LIN {X 0,Y 179.464,Z 996.724,A -85,B 0,C 180,E1 20811.906,E2 20811.906} C_VEL
LIN {X 0,Y 188.427,Z 983.505,A -85,B 0,C 180,E1 20823.22,E2 20823.22} C_VEL
LIN {X 0,Y 202.809,Z 964.358,A -85,B 0,C 180,E1 20832.94,E2 20832.94} C_VEL
LIN {X 0,Y 221.661,Z 939.292,A -85,B 0,C 180,E1 20840.906,E2 20840.906} C_VEL
LIN {X 0,Y 224.713,Z 937.25,A -85,B 0,C 180,E1 20842.19,E2 20842.19} C_VEL
LIN {X 0,Y 206.607,Z 940.656,A -85,B 0,C 180,E1 20849.15,E2 20849.15} C_VEL
LIN {X 0,Y 193.54,Z 940.036,A -85,B 0,C 180,E1 20856.986,E2 20856.986} C_VEL
LIN {X 0,Y 184.714,Z 935.319,A -85,B 0,C 180,E1 20865.776,E2 20865.776} C_VEL
LIN {X 0,Y 180.026,Z 924.585,A -85,B 0,C 180,E1 20876.395,E2 20876.395} C_VEL
LIN {X 0,Y 191.865,Z 914.932,A -85,B 0,C 180,E1 20893.704,E2 20893.704} C_VEL
LIN {X 0,Y 212.483,Z 904.44,A -85,B 0,C 180,E1 20904.008,E2 20904.008} C_VEL
LIN {X 0,Y 233.891,Z 893.022,A -85,B 0,C 180,E1 20910.12,E2 20910.12} C_VEL
LIN {X 0,Y 248.033,Z 884.252,A -85,B 0,C 180,E1 20912.881,E2 20912.881} C_VEL
LIN {X 0,Y 238.457,Z 902.02,A -85,B 0,C 180,E1 20915.584,E2 20915.584} C_VEL
LIN {X 0,Y 228.286,Z 914.831,A -85,B 0,C 180,E1 20917.177,E2 20917.177} C_VEL
LIN {X 0,Y 217.808,Z 926.758,A -85,B 0,C 180,E1 20919.046,E2 20919.046} C_VEL
LIN {X 0,Y 200.214,Z 949.54,A -85,B 0,C 180,E1 20926.435,E2 20926.435} C_VEL
LIN {X 0,Y 185.842,Z 966.385,A -85,B 0,C 180,E1 20935.229,E2 20935.229} C_VEL
LIN {X 0,Y 174.431,Z 979.636,A -85,B 0,C 180,E1 20947.008,E2 20947.008} C_VEL
LIN {X 0,Y 169.075,Z 986.655,A -85,B 0,C 180,E1 20959.683,E2 20959.683} C_VEL
LIN {X 0,Y 168.279,Z 988.372,A -85,B 0,C 180,E1 20970.001,E2 20970.001} C_VEL
LIN {X 0,Y 169.698,Z 985.642,A -85,B 0,C 180,E1 20982.889,E2 20982.889} C_VEL
LIN {X 0,Y 176.265,Z 977.344,A -85,B 0,C 180,E1 20995.436,E2 20995.436} C_VEL
LIN {X 0,Y 188.345,Z 963.517,A -85,B 0,C 180,E1 21006.483,E2 21006.483} C_VEL
LIN {X 0,Y 204.243,Z 944.465,A -85,B 0,C 180,E1 21015.398,E2 21015.398} C_VEL
LIN {X 0,Y 221.705,Z 921.014,A -85,B 0,C 180,E1 21022.202,E2 21022.202} C_VEL
LIN {X 0,Y 239.619,Z 892.347,A -85,B 0,C 180,E1 21027.459,E2 21027.459} C_VEL
LIN {X 0,Y 247.476,Z 877.194,A -85,B 0,C 180,E1 21029.455,E2 21029.455} C_VEL
LIN {X 0,Y 247.461,Z 861.301,A -85,B 0,C 180,E1 21034.633,E2 21034.633} C_VEL
LIN {X 0,Y 245.563,Z 845.485,A -85,B 0,C 180,E1 21041.277,E2 21041.277} C_VEL
LIN {X 0,Y 243.44,Z 835.366,A -85,B 0,C 180,E1 21047.419,E2 21047.419} C_VEL
LIN {X 0,Y 242.204,Z 826.553,A -85,B 0,C 180,E1 21056.408,E2 21056.408} C_VEL
LIN {X 0,Y 242.269,Z 825.858,A -85,B 0,C 180,E1 21060.576,E2 21060.576} C_VEL
LIN {X 0,Y 242.778,Z 829.253,A -85,B 0,C 180,E1 21065.961,E2 21065.961} C_VEL
LIN {X 0,Y 244.587,Z 835.008,A -85,B 0,C 180,E1 21071.486,E2 21071.486} C_VEL
LIN {X 0,Y 247.754,Z 845.599,A -85,B 0,C 180,E1 21077.783,E2 21077.783} C_VEL
LIN {X 0,Y 251.247,Z 862.741,A -85,B 0,C 180,E1 21084.577,E2 21084.577} C_VEL
LIN {X 0,Y 252.298,Z 874.194,A -85,B 0,C 180,E1 21088.056,E2 21088.056} C_VEL
LIN {X 0,Y 235.917,Z 906.866,A -85,B 0,C 180,E1 21091.747,E2 21091.747} C_VEL
LIN {X 0,Y 217.801,Z 935.609,A -85,B 0,C 180,E1 21096.922,E2 21096.922} C_VEL
LIN {X 0,Y 199.968,Z 960.052,A -85,B 0,C 180,E1 21104.002,E2 21104.002} C_VEL
LIN {X 0,Y 184.115,Z 979.936,A -85,B 0,C 180,E1 21113.4,E2 21113.4} C_VEL
LIN {X 0,Y 173.683,Z 993.599,A -85,B 0,C 180,E1 21124.158,E2 21124.158} C_VEL
LIN {X 0,Y 168.628,Z 1002.638,A -85,B 0,C 180,E1 21137.027,E2 21137.027} C_VEL
LIN {X 0,Y 167.979,Z 1005.154,A -85,B 0,C 180,E1 21144.828,E2 21144.828} C_VEL
LIN {X 0,Y 168.272,Z 1005.706,A -85,B 0,C 180,E1 21149.999,E2 21149.999} C_VEL
LIN {X 0,Y 168.316,Z 1003.73,A -85,B 0,C 180,E1 21160.364,E2 21160.364} C_VEL
LIN {X 0,Y 171.974,Z 996.308,A -85,B 0,C 180,E1 21172.913,E2 21172.913} C_VEL
LIN {X 0,Y 181.684,Z 983.091,A -85,B 0,C 180,E1 21184.622,E2 21184.622} C_VEL
LIN {X 0,Y 196.959,Z 963.946,A -85,B 0,C 180,E1 21194.544,E2 21194.544} C_VEL
LIN {X 0,Y 214.742,Z 941.387,A -85,B 0,C 180,E1 21201.936,E2 21201.936} C_VEL
LIN {X 0,Y 212.168,Z 941.574,A -85,B 0,C 180,E1 21203.228,E2 21203.228} C_VEL
LIN {X 0,Y 192.759,Z 942.674,A -85,B 0,C 180,E1 21211.895,E2 21211.895} C_VEL
LIN {X 0,Y 178.981,Z 937.997,A -85,B 0,C 180,E1 21222.79,E2 21222.79} C_VEL
LIN {X 0,Y 174.357,Z 932.944,A -85,B 0,C 180,E1 21230.01,E2 21230.01} C_VEL
LIN {X 0,Y 183.786,Z 922.038,A -85,B 0,C 180,E1 21252.128,E2 21252.128} C_VEL
LIN {X 0,Y 205.4,Z 911.59,A -85,B 0,C 180,E1 21263.927,E2 21263.927} C_VEL
LIN {X 0,Y 229.608,Z 899.619,A -85,B 0,C 180,E1 21270.992,E2 21270.992} C_VEL
LIN {X 0,Y 237.877,Z 894.762,A -85,B 0,C 180,E1 21272.576,E2 21272.576} C_VEL
LIN {X 0,Y 228.28,Z 911.475,A -85,B 0,C 180,E1 21275.66,E2 21275.66} C_VEL
LIN {X 0,Y 217.808,Z 926.758,A -85,B 0,C 180,E1 21279.046,E2 21279.046} C_VEL
LIN {X 0,Y 207.123,Z 937.885,A -85,B 0,C 180,E1 21281.311,E2 21281.311} C_VEL
LIN {X 0,Y 196.269,Z 947.941,A -85,B 0,C 180,E1 21283.983,E2 21283.983} C_VEL
LIN {X 0,Y 180.439,Z 965.598,A -85,B 0,C 180,E1 21292.966,E2 21292.966} C_VEL
LIN {X 0,Y 168.599,Z 978.34,A -85,B 0,C 180,E1 21303.922,E2 21303.922} C_VEL
LIN {X 0,Y 161.955,Z 986.12,A -85,B 0,C 180,E1 21316.485,E2 21316.485} C_VEL
LIN {X 0,Y 160.382,Z 988.779,A -85,B 0,C 180,E1 21330.001,E2 21330.001} C_VEL
LIN {X 0,Y 161.962,Z 986.052,A -85,B 0,C 180,E1 21343.516,E2 21343.516} C_VEL
LIN {X 0,Y 169.086,Z 977.756,A -85,B 0,C 180,E1 21356.599,E2 21356.599} C_VEL
LIN {X 0,Y 181.946,Z 963.931,A -85,B 0,C 180,E1 21367.988,E2 21367.988} C_VEL
LIN {X 0,Y 198.97,Z 944.564,A -85,B 0,C 180,E1 21377.152,E2 21377.152} C_VEL
LIN {X 0,Y 217.234,Z 921.012,A -85,B 0,C 180,E1 21383.95,E2 21383.95} C_VEL
LIN {X 0,Y 235.808,Z 892.059,A -85,B 0,C 180,E1 21389.19,E2 21389.19} C_VEL
LIN {X 0,Y 242.442,Z 879.285,A -85,B 0,C 180,E1 21390.966,E2 21390.966} C_VEL
LIN {X 0,Y 242.488,Z 862.032,A -85,B 0,C 180,E1 21397.193,E2 21397.193} C_VEL
LIN {X 0,Y 241.095,Z 848.707,A -85,B 0,C 180,E1 21403.571,E2 21403.571} C_VEL
LIN {X 0,Y 239.529,Z 838.708,A -85,B 0,C 180,E1 21410.9,E2 21410.9} C_VEL
LIN {X 0,Y 239.279,Z 834.165,A -85,B 0,C 180,E1 21416.364,E2 21416.364} C_VEL
LIN {X 0,Y 239.517,Z 833.081,A -85,B 0,C 180,E1 21419.992,E2 21419.992} C_VEL
LIN {X 0,Y 239.769,Z 836.262,A -85,B 0,C 180,E1 21425.427,E2 21425.427} C_VEL
LIN {X 0,Y 241.615,Z 842.867,A -85,B 0,C 180,E1 21431.742,E2 21431.742} C_VEL
LIN {X 0,Y 244.491,Z 855.04,A -85,B 0,C 180,E1 21438.617,E2 21438.617} C_VEL
LIN {X 0,Y 246.818,Z 871.391,A -85,B 0,C 180,E1 21444.934,E2 21444.934} C_VEL
LIN {X 0,Y 246.894,Z 877.599,A -85,B 0,C 180,E1 21446.755,E2 21446.755} C_VEL
LIN {X 0,Y 230.237,Z 908.983,A -85,B 0,C 180,E1 21450.415,E2 21450.415} C_VEL
LIN {X 0,Y 211.524,Z 937.345,A -85,B 0,C 180,E1 21455.677,E2 21455.677} C_VEL
LIN {X 0,Y 192.285,Z 962.191,A -85,B 0,C 180,E1 21463.249,E2 21463.249} C_VEL
LIN {X 0,Y 176.106,Z 981.296,A -85,B 0,C 180,E1 21472.998,E2 21472.998} C_VEL
LIN {X 0,Y 164.763,Z 995.485,A -85,B 0,C 180,E1 21485.503,E2 21485.503} C_VEL
LIN {X 0,Y 160.816,Z 1002.224,A -85,B 0,C 180,E1 21496.385,E2 21496.385} C_VEL
LIN {X 0,Y 160.089,Z 1004.746,A -85,B 0,C 180,E1 21504.572,E2 21504.572} C_VEL
LIN {X 0,Y 160.367,Z 1005.299,A -85,B 0,C 180,E1 21509.999,E2 21509.999} C_VEL
LIN {X 0,Y 160.452,Z 1003.318,A -85,B 0,C 180,E1 21520.878,E2 21520.878} C_VEL
LIN {X 0,Y 163.73,Z 997.099,A -85,B 0,C 180,E1 21532.408,E2 21532.408} C_VEL
LIN {X 0,Y 173.308,Z 984.718,A -85,B 0,C 180,E1 21544.648,E2 21544.648} C_VEL
LIN {X 0,Y 189.278,Z 965.914,A -85,B 0,C 180,E1 21555.271,E2 21555.271} C_VEL
LIN {X 0,Y 205.092,Z 946.288,A -85,B 0,C 180,E1 21562.062,E2 21562.062} C_VEL
LIN {X 0,Y 204.779,Z 945.296,A -85,B 0,C 180,E1 21562.662,E2 21562.662} C_VEL
LIN {X 0,Y 179.561,Z 943.046,A -85,B 0,C 180,E1 21574.911,E2 21574.911} C_VEL
LIN {X 0,Y 167.76,Z 936.904,A -85,B 0,C 180,E1 21593.109,E2 21593.109} C_VEL
LIN {X 0,Y 183.267,Z 925.022,A -85,B 0,C 180,E1 21616.377,E2 21616.377} C_VEL
LIN {X 0,Y 206.574,Z 914.687,A -85,B 0,C 180,E1 21626.877,E2 21626.877} C_VEL
LIN {X 0,Y 228.196,Z 904.473,A -85,B 0,C 180,E1 21632.514,E2 21632.514} C_VEL
LIN {X 0,Y 210.055,Z 930.89,A -85,B 0,C 180,E1 21638.384,E2 21638.384} C_VEL
LIN {X 0,Y 196.269,Z 947.941,A -85,B 0,C 180,E1 21643.983,E2 21643.983} C_VEL
LIN {X 0,Y 185.45,Z 957.053,A -85,B 0,C 180,E1 21647.123,E2 21647.123} C_VEL
LIN {X 0,Y 174.986,Z 965.107,A -85,B 0,C 180,E1 21650.773,E2 21650.773} C_VEL
LIN {X 0,Y 161.911,Z 978.288,A -85,B 0,C 180,E1 21662.124,E2 21662.124} C_VEL
LIN {X 0,Y 154.238,Z 986.529,A -85,B 0,C 180,E1 21675.794,E2 21675.794} C_VEL
LIN {X 0,Y 152.486,Z 989.186,A -85,B 0,C 180,E1 21690.001,E2 21690.001} C_VEL
LIN {X 0,Y 153.487,Z 987.424,A -85,B 0,C 180,E1 21701.38,E2 21701.38} C_VEL
LIN {X 0,Y 159.51,Z 980.709,A -85,B 0,C 180,E1 21714.713,E2 21714.713} C_VEL
LIN {X 0,Y 171.409,Z 968.7,A -85,B 0,C 180,E1 21726.602,E2 21726.602} C_VEL
LIN {X 0,Y 188.084,Z 951.162,A -85,B 0,C 180,E1 21736.429,E2 21736.429} C_VEL
LIN {X 0,Y 206.516,Z 929.398,A -85,B 0,C 180,E1 21743.754,E2 21743.754} C_VEL
LIN {X 0,Y 226.287,Z 901.602,A -85,B 0,C 180,E1 21749.483,E2 21749.483} C_VEL
LIN {X 0,Y 236.896,Z 883.541,A -85,B 0,C 180,E1 21752.058,E2 21752.058} C_VEL
LIN {X 0,Y 237.815,Z 870.108,A -85,B 0,C 180,E1 21756.907,E2 21756.907} C_VEL
LIN {X 0,Y 237.346,Z 856.865,A -85,B 0,C 180,E1 21763.117,E2 21763.117} C_VEL
LIN {X 0,Y 236.3,Z 847.248,A -85,B 0,C 180,E1 21769.843,E2 21769.843} C_VEL
LIN {X 0,Y 236.177,Z 841.656,A -85,B 0,C 180,E1 21776.316,E2 21776.316} C_VEL
LIN {X 0,Y 236.562,Z 840.453,A -85,B 0,C 180,E1 21779.992,E2 21779.992} C_VEL
LIN {X 0,Y 237.055,Z 845.156,A -85,B 0,C 180,E1 21787.33,E2 21787.33} C_VEL
LIN {X 0,Y 239.179,Z 854.781,A -85,B 0,C 180,E1 21794.659,E2 21794.659} C_VEL
LIN {X 0,Y 241.299,Z 869.107,A -85,B 0,C 180,E1 21801.41,E2 21801.41} C_VEL
LIN {X 0,Y 241.687,Z 880.713,A -85,B 0,C 180,E1 21805.414,E2 21805.414} C_VEL
LIN {X 0,Y 224.968,Z 910.673,A -85,B 0,C 180,E1 21808.962,E2 21808.962} C_VEL
LIN {X 0,Y 205.494,Z 938.877,A -85,B 0,C 180,E1 21814.311,E2 21814.311} C_VEL
LIN {X 0,Y 185.623,Z 963.12,A -85,B 0,C 180,E1 21821.988,E2 21821.988} C_VEL
LIN {X 0,Y 169.679,Z 980.877,A -85,B 0,C 180,E1 21831.344,E2 21831.344} C_VEL
LIN {X 0,Y 157.4,Z 995.119,A -85,B 0,C 180,E1 21844.349,E2 21844.349} C_VEL
LIN {X 0,Y 152.595,Z 1002.885,A -85,B 0,C 180,E1 21858.553,E2 21858.553} C_VEL
LIN {X 0,Y 152.46,Z 1004.892,A -85,B 0,C 180,E1 21869.999,E2 21869.999} C_VEL
LIN {X 0,Y 152.598,Z 1002.907,A -85,B 0,C 180,E1 21881.445,E2 21881.445} C_VEL
LIN {X 0,Y 157.439,Z 995.164,A -85,B 0,C 180,E1 21895.642,E2 21895.642} C_VEL
LIN {X 0,Y 167.967,Z 982.916,A -85,B 0,C 180,E1 21907.315,E2 21907.315} C_VEL
LIN {X 0,Y 184.685,Z 964.344,A -85,B 0,C 180,E1 21917.547,E2 21917.547} C_VEL
LIN {X 0,Y 195.462,Z 951.703,A -85,B 0,C 180,E1 21922.156,E2 21922.156} C_VEL
LIN {X 0,Y 196.158,Z 950.097,A -85,B 0,C 180,E1 21922.851,E2 21922.851} C_VEL
LIN {X 0,Y 173.76,Z 947.877,A -85,B 0,C 180,E1 21934.185,E2 21934.185} C_VEL
LIN {X 0,Y 162.4,Z 943.173,A -85,B 0,C 180,E1 21949.266,E2 21949.266} C_VEL
LIN {X 0,Y 171.847,Z 933.069,A -85,B 0,C 180,E1 21972.719,E2 21972.719} C_VEL
LIN {X 0,Y 196.729,Z 922.491,A -85,B 0,C 180,E1 21986.095,E2 21986.095} C_VEL
LIN {X 0,Y 218.362,Z 913.089,A -85,B 0,C 180,E1 21992.239,E2 21992.239} C_VEL
LIN {X 0,Y 200.388,Z 937.238,A -85,B 0,C 180,E1 21998.381,E2 21998.381} C_VEL
LIN {X 0,Y 181.84,Z 957.971,A -85,B 0,C 180,E1 22006.613,E2 22006.613} C_VEL
LIN {X 0,Y 174.986,Z 965.107,A -85,B 0,C 180,E1 22010.773,E2 22010.773} C_VEL
LIN {X 0,Y 164.934,Z 972.156,A -85,B 0,C 180,E1 22015.005,E2 22015.005} C_VEL
LIN {X 0,Y 155.629,Z 978.011,A -85,B 0,C 180,E1 22019.894,E2 22019.894} C_VEL
LIN {X 0,Y 147.717,Z 985.786,A -85,B 0,C 180,E1 22032.092,E2 22032.092} C_VEL
LIN {X 0,Y 144.652,Z 989.15,A -85,B 0,C 180,E1 22043.993,E2 22043.993} C_VEL
LIN {X 0,Y 144.616,Z 989.591,A -85,B 0,C 180,E1 22050.001,E2 22050.001} C_VEL
LIN {X 0,Y 146.565,Z 986.871,A -85,B 0,C 180,E1 22064.968,E2 22064.968} C_VEL
LIN {X 0,Y 154.948,Z 978.58,A -85,B 0,C 180,E1 22079.248,E2 22079.248} C_VEL
LIN {X 0,Y 169.042,Z 965.289,A -85,B 0,C 180,E1 22090.959,E2 22090.959} C_VEL
LIN {X 0,Y 187.343,Z 946.622,A -85,B 0,C 180,E1 22100.264,E2 22100.264} C_VEL
LIN {X 0,Y 207.545,Z 922.725,A -85,B 0,C 180,E1 22107.296,E2 22107.296} C_VEL
LIN {X 0,Y 227.348,Z 894.114,A -85,B 0,C 180,E1 22112.445,E2 22112.445} C_VEL
LIN {X 0,Y 231.835,Z 886.48,A -85,B 0,C 180,E1 22113.46,E2 22113.46} C_VEL
LIN {X 0,Y 233.119,Z 872.263,A -85,B 0,C 180,E1 22119.063,E2 22119.063} C_VEL
LIN {X 0,Y 233.03,Z 861.052,A -85,B 0,C 180,E1 22124.928,E2 22124.928} C_VEL
LIN {X 0,Y 232.573,Z 853.149,A -85,B 0,C 180,E1 22131.178,E2 22131.178} C_VEL
LIN {X 0,Y 232.869,Z 849.045,A -85,B 0,C 180,E1 22136.264,E2 22136.264} C_VEL
LIN {X 0,Y 233.312,Z 847.701,A -85,B 0,C 180,E1 22139.992,E2 22139.992} C_VEL
LIN {X 0,Y 233.72,Z 852.568,A -85,B 0,C 180,E1 22147.436,E2 22147.436} C_VEL
LIN {X 0,Y 235.399,Z 862.555,A -85,B 0,C 180,E1 22154.899,E2 22154.899} C_VEL
LIN {X 0,Y 236.663,Z 875.873,A -85,B 0,C 180,E1 22161.143,E2 22161.143} C_VEL
LIN {X 0,Y 236.88,Z 883.071,A -85,B 0,C 180,E1 22163.887,E2 22163.887} C_VEL
LIN {X 0,Y 218.289,Z 914.772,A -85,B 0,C 180,E1 22167.825,E2 22167.825} C_VEL
LIN {X 0,Y 198.808,Z 941.195,A -85,B 0,C 180,E1 22173.096,E2 22173.096} C_VEL
LIN {X 0,Y 179.277,Z 963.802,A -85,B 0,C 180,E1 22180.526,E2 22180.526} C_VEL
LIN {X 0,Y 161.73,Z 982.238,A -85,B 0,C 180,E1 22190.807,E2 22190.807} C_VEL
LIN {X 0,Y 149.255,Z 995.707,A -85,B 0,C 180,E1 22204.459,E2 22204.459} C_VEL
LIN {X 0,Y 144.752,Z 1002.472,A -85,B 0,C 180,E1 22217.924,E2 22217.924} C_VEL
LIN {X 0,Y 144.579,Z 1004.486,A -85,B 0,C 180,E1 22229.999,E2 22229.999} C_VEL
LIN {X 0,Y 144.76,Z 1002.495,A -85,B 0,C 180,E1 22242.074,E2 22242.074} C_VEL
LIN {X 0,Y 150.179,Z 994.748,A -85,B 0,C 180,E1 22256.98,E2 22256.98} C_VEL
LIN {X 0,Y 161.732,Z 982.325,A -85,B 0,C 180,E1 22269.191,E2 22269.191} C_VEL
LIN {X 0,Y 179.27,Z 963.928,A -85,B 0,C 180,E1 22279.474,E2 22279.474} C_VEL
LIN {X 0,Y 186.444,Z 956.036,A -85,B 0,C 180,E1 22282.505,E2 22282.505} C_VEL
LIN {X 0,Y 187.012,Z 954.653,A -85,B 0,C 180,E1 22283.226,E2 22283.226} C_VEL
LIN {X 0,Y 162.395,Z 951.418,A -85,B 0,C 180,E1 22298.117,E2 22298.117} C_VEL
LIN {X 0,Y 159.056,Z 941.814,A -85,B 0,C 180,E1 22325.474,E2 22325.474} C_VEL
LIN {X 0,Y 179.884,Z 932.455,A -85,B 0,C 180,E1 22342.201,E2 22342.201} C_VEL
LIN {X 0,Y 208.032,Z 921.507,A -85,B 0,C 180,E1 22351.984,E2 22351.984} C_VEL
LIN {X 0,Y 206.688,Z 924.018,A -85,B 0,C 180,E1 22352.863,E2 22352.863} C_VEL
LIN {X 0,Y 186.674,Z 947.564,A -85,B 0,C 180,E1 22359.962,E2 22359.962} C_VEL
LIN {X 0,Y 168.244,Z 966.111,A -85,B 0,C 180,E1 22369.454,E2 22369.454} C_VEL
LIN {X 0,Y 155.629,Z 978.011,A -85,B 0,C 180,E1 22379.894,E2 22379.894} C_VEL
LIN {X 0,Y 147.326,Z 982.756,A -85,B 0,C 180,E1 22385.447,E2 22385.447} C_VEL
LIN {X 0,Y 139.907,Z 986.406,A -85,B 0,C 180,E1 22391.655,E2 22391.655} C_VEL
LIN {X 0,Y 136.603,Z 989.825,A -85,B 0,C 180,E1 22406.151,E2 22406.151} C_VEL
LIN {X 0,Y 136.849,Z 989.527,A -85,B 0,C 180,E1 22416.353,E2 22416.353} C_VEL
LIN {X 0,Y 141.686,Z 984.662,A -85,B 0,C 180,E1 22431.965,E2 22431.965} C_VEL
LIN {X 0,Y 153.773,Z 974.013,A -85,B 0,C 180,E1 22446.213,E2 22446.213} C_VEL
LIN {X 0,Y 171.774,Z 957.505,A -85,B 0,C 180,E1 22457.58,E2 22457.58} C_VEL
LIN {X 0,Y 192.248,Z 936.331,A -85,B 0,C 180,E1 22465.788,E2 22465.788} C_VEL
LIN {X 0,Y 213.412,Z 909.87,A -85,B 0,C 180,E1 22471.841,E2 22471.841} C_VEL
LIN {X 0,Y 226.798,Z 889.535,A -85,B 0,C 180,E1 22474.897,E2 22474.897} C_VEL
LIN {X 0,Y 228.562,Z 875.02,A -85,B 0,C 180,E1 22481.151,E2 22481.151} C_VEL
LIN {X 0,Y 228.863,Z 864.082,A -85,B 0,C 180,E1 22487.746,E2 22487.746} C_VEL
LIN {X 0,Y 229.255,Z 856.286,A -85,B 0,C 180,E1 22496.205,E2 22496.205} C_VEL
LIN {X 0,Y 229.858,Z 854.841,A -85,B 0,C 180,E1 22499.992,E2 22499.992} C_VEL
LIN {X 0,Y 230.083,Z 859.858,A -85,B 0,C 180,E1 22507.554,E2 22507.554} C_VEL
LIN {X 0,Y 231.193,Z 869.157,A -85,B 0,C 180,E1 22514.548,E2 22514.548} C_VEL
LIN {X 0,Y 231.79,Z 882.739,A -85,B 0,C 180,E1 22520.998,E2 22520.998} C_VEL
LIN {X 0,Y 231.767,Z 886.188,A -85,B 0,C 180,E1 22522.359,E2 22522.359} C_VEL
LIN {X 0,Y 212.418,Z 917.532,A -85,B 0,C 180,E1 22526.433,E2 22526.433} C_VEL
LIN {X 0,Y 191.785,Z 944.013,A -85,B 0,C 180,E1 22531.93,E2 22531.93} C_VEL
LIN {X 0,Y 170.651,Z 966.946,A -85,B 0,C 180,E1 22540.069,E2 22540.069} C_VEL
LIN {X 0,Y 153.805,Z 983.44,A -85,B 0,C 180,E1 22550.216,E2 22550.216} C_VEL
LIN {X 0,Y 141.092,Z 996.292,A -85,B 0,C 180,E1 22564.579,E2 22564.579} C_VEL
LIN {X 0,Y 136.954,Z 1002.06,A -85,B 0,C 180,E1 22577.225,E2 22577.225} C_VEL
LIN {X 0,Y 136.67,Z 1004.078,A -85,B 0,C 180,E1 22589.999,E2 22589.999} C_VEL
LIN {X 0,Y 136.965,Z 1002.084,A -85,B 0,C 180,E1 22602.772,E2 22602.772} C_VEL
LIN {X 0,Y 142.996,Z 994.332,A -85,B 0,C 180,E1 22618.454,E2 22618.454} C_VEL
LIN {X 0,Y 155.518,Z 981.909,A -85,B 0,C 180,E1 22631.083,E2 22631.083} C_VEL
LIN {X 0,Y 174.115,Z 963.517,A -85,B 0,C 180,E1 22641.501,E2 22641.501} C_VEL
LIN {X 0,Y 178.06,Z 959.012,A -85,B 0,C 180,E1 22643.487,E2 22643.487} C_VEL
LIN {X 0,Y 152.166,Z 954.451,A -85,B 0,C 180,E1 22662.646,E2 22662.646} C_VEL
LIN {X 0,Y 156.961,Z 944.359,A -85,B 0,C 180,E1 22691.136,E2 22691.136} C_VEL
LIN {X 0,Y 184.436,Z 933.953,A -85,B 0,C 180,E1 22707.399,E2 22707.399} C_VEL
LIN {X 0,Y 198.509,Z 928.804,A -85,B 0,C 180,E1 22711.81,E2 22711.81} C_VEL
LIN {X 0,Y 179.736,Z 949.883,A -85,B 0,C 180,E1 22718.812,E2 22718.812} C_VEL
LIN {X 0,Y 160.547,Z 968.024,A -85,B 0,C 180,E1 22728.689,E2 22728.689} C_VEL
LIN {X 0,Y 146.076,Z 980.815,A -85,B 0,C 180,E1 22741.436,E2 22741.436} C_VEL
LIN {X 0,Y 139.907,Z 986.406,A -85,B 0,C 180,E1 22751.655,E2 22751.655} C_VEL
LIN {X 0,Y 135.51,Z 988.359,A -85,B 0,C 180,E1 22756.725,E2 22756.725} C_VEL
LIN {X 0,Y 128.693,Z 990.217,A -85,B 0,C 180,E1 22765.518,E2 22765.518} C_VEL
LIN {X 0,Y 128.675,Z 990.129,A -85,B 0,C 180,E1 22765.763,E2 22765.763} C_VEL
LIN {X 0,Y 128.981,Z 989.935,A -85,B 0,C 180,E1 22776.742,E2 22776.742} C_VEL
LIN {X 0,Y 134.31,Z 985.074,A -85,B 0,C 180,E1 22793.239,E2 22793.239} C_VEL
LIN {X 0,Y 147.375,Z 974.427,A -85,B 0,C 180,E1 22808.057,E2 22808.057} C_VEL
LIN {X 0,Y 165.12,Z 959.167,A -85,B 0,C 180,E1 22818.973,E2 22818.973} C_VEL
LIN {X 0,Y 186.229,Z 938.477,A -85,B 0,C 180,E1 22827.277,E2 22827.277} C_VEL
LIN {X 0,Y 207.423,Z 913.44,A -85,B 0,C 180,E1 22833.191,E2 22833.191} C_VEL
LIN {X 0,Y 221.817,Z 892.731,A -85,B 0,C 180,E1 22836.385,E2 22836.385} C_VEL
LIN {X 0,Y 223.896,Z 880.01,A -85,B 0,C 180,E1 22842.201,E2 22842.201} C_VEL
LIN {X 0,Y 224.72,Z 870.387,A -85,B 0,C 180,E1 22848.33,E2 22848.33} C_VEL
LIN {X 0,Y 225.454,Z 863.439,A -85,B 0,C 180,E1 22856.141,E2 22856.141} C_VEL
LIN {X 0,Y 226.232,Z 861.897,A -85,B 0,C 180,E1 22859.991,E2 22859.991} C_VEL
LIN {X 0,Y 226.221,Z 867.042,A -85,B 0,C 180,E1 22867.684,E2 22867.684} C_VEL
LIN {X 0,Y 226.857,Z 876.189,A -85,B 0,C 180,E1 22874.485,E2 22874.485} C_VEL
LIN {X 0,Y 226.719,Z 889.254,A -85,B 0,C 180,E1 22880.777,E2 22880.777} C_VEL
LIN {X 0,Y 207.433,Z 919.235,A -85,B 0,C 180,E1 22884.79,E2 22884.79} C_VEL
LIN {X 0,Y 184.852,Z 946.695,A -85,B 0,C 180,E1 22890.678,E2 22890.678} C_VEL
LIN {X 0,Y 163.188,Z 968.741,A -85,B 0,C 180,E1 22899.007,E2 22899.007} C_VEL
LIN {X 0,Y 144.184,Z 986.17,A -85,B 0,C 180,E1 22910.944,E2 22910.944} C_VEL
LIN {X 0,Y 132.118,Z 997.705,A -85,B 0,C 180,E1 22926.42,E2 22926.42} C_VEL
LIN {X 0,Y 129.144,Z 1001.647,A -85,B 0,C 180,E1 22936.438,E2 22936.438} C_VEL
LIN {X 0,Y 128.766,Z 1003.671,A -85,B 0,C 180,E1 22949.999,E2 22949.999} C_VEL
LIN {X 0,Y 129.157,Z 1001.672,A -85,B 0,C 180,E1 22963.559,E2 22963.559} C_VEL
LIN {X 0,Y 135.938,Z 993.917,A -85,B 0,C 180,E1 22980.079,E2 22980.079} C_VEL
LIN {X 0,Y 151.386,Z 979.714,A -85,B 0,C 180,E1 22994.434,E2 22994.434} C_VEL
LIN {X 0,Y 169.199,Z 963.105,A -85,B 0,C 180,E1 23003.645,E2 23003.645} C_VEL
LIN {X 0,Y 145.849,Z 958.831,A -85,B 0,C 180,E1 23021.869,E2 23021.869} C_VEL
LIN {X 0,Y 150.548,Z 949.059,A -85,B 0,C 180,E1 23051.616,E2 23051.616} C_VEL
LIN {X 0,Y 177.657,Z 939.448,A -85,B 0,C 180,E1 23067.963,E2 23067.963} C_VEL
LIN {X 0,Y 188.32,Z 935.88,A -85,B 0,C 180,E1 23071.492,E2 23071.492} C_VEL
LIN {X 0,Y 182.507,Z 942.681,A -85,B 0,C 180,E1 23073.943,E2 23073.943} C_VEL
LIN {X 0,Y 162.963,Z 961.221,A -85,B 0,C 180,E1 23081.989,E2 23081.989} C_VEL
LIN {X 0,Y 145.625,Z 975.867,A -85,B 0,C 180,E1 23093.286,E2 23093.286} C_VEL
LIN {X 0,Y 134.29,Z 985.155,A -85,B 0,C 180,E1 23106.759,E2 23106.759} C_VEL
LIN {X 0,Y 130.21,Z 988.697,A -85,B 0,C 180,E1 23116.553,E2 23116.553} C_VEL
LIN {X 0,Y 128.675,Z 990.129,A -85,B 0,C 180,E1 23125.763,E2 23125.763} C_VEL
LIN {X 0,Y 126.051,Z 990.508,A -85,B 0,C 180,E1 23131.529,E2 23131.529} C_VEL
LIN {X 0,Y 121.769,Z 989.554,A -85,B 0,C 180,E1 23141.583,E2 23141.583} C_VEL
LIN {X 0,Y 129.173,Z 983.844,A -85,B 0,C 180,E1 23157.961,E2 23157.961} C_VEL
LIN {X 0,Y 143.452,Z 973.016,A -85,B 0,C 180,E1 23171.744,E2 23171.744} C_VEL
LIN {X 0,Y 163.588,Z 956.457,A -85,B 0,C 180,E1 23182.717,E2 23182.717} C_VEL
LIN {X 0,Y 186.107,Z 934.648,A -85,B 0,C 180,E1 23190.622,E2 23190.622} C_VEL
LIN {X 0,Y 208.411,Z 907.948,A -85,B 0,C 180,E1 23196.183,E2 23196.183} C_VEL
LIN {X 0,Y 217.033,Z 895.795,A -85,B 0,C 180,E1 23197.956,E2 23197.956} C_VEL
LIN {X 0,Y 219.417,Z 883.746,A -85,B 0,C 180,E1 23203.969,E2 23203.969} C_VEL
LIN {X 0,Y 220.526,Z 875.308,A -85,B 0,C 180,E1 23210.108,E2 23210.108} C_VEL
LIN {X 0,Y 221.481,Z 870.477,A -85,B 0,C 180,E1 23216.071,E2 23216.071} C_VEL
LIN {X 0,Y 222.332,Z 868.846,A -85,B 0,C 180,E1 23219.991,E2 23219.991} C_VEL
LIN {X 0,Y 222.141,Z 874.179,A -85,B 0,C 180,E1 23227.826,E2 23227.826} C_VEL
LIN {X 0,Y 222.299,Z 883.918,A -85,B 0,C 180,E1 23234.895,E2 23234.895} C_VEL
LIN {X 0,Y 221.723,Z 892.684,A -85,B 0,C 180,E1 23239.218,E2 23239.218} C_VEL
LIN {X 0,Y 201.848,Z 921.906,A -85,B 0,C 180,E1 23243.234,E2 23243.234} C_VEL
LIN {X 0,Y 179.438,Z 947.758,A -85,B 0,C 180,E1 23248.901,E2 23248.901} C_VEL
LIN {X 0,Y 156.974,Z 969.428,A -85,B 0,C 180,E1 23257.272,E2 23257.272} C_VEL
LIN {X 0,Y 137.991,Z 985.753,A -85,B 0,C 180,E1 23268.825,E2 23268.825} C_VEL
LIN {X 0,Y 124.74,Z 997.287,A -85,B 0,C 180,E1 23284.932,E2 23284.932} C_VEL
LIN {X 0,Y 121.356,Z 1001.234,A -85,B 0,C 180,E1 23295.549,E2 23295.549} C_VEL
LIN {X 0,Y 120.868,Z 1003.265,A -85,B 0,C 180,E1 23309.999,E2 23309.999} C_VEL
LIN {X 0,Y 121.372,Z 1001.259,A -85,B 0,C 180,E1 23324.447,E2 23324.447} C_VEL
LIN {X 0,Y 128.982,Z 993.5,A -85,B 0,C 180,E1 23341.886,E2 23341.886} C_VEL
LIN {X 0,Y 145.682,Z 979.298,A -85,B 0,C 180,E1 23356.677,E2 23356.677} C_VEL
LIN {X 0,Y 159.19,Z 967.57,A -85,B 0,C 180,E1 23363.706,E2 23363.706} C_VEL
LIN {X 0,Y 158.338,Z 966.593,A -85,B 0,C 180,E1 23365.006,E2 23365.006} C_VEL
LIN {X 0,Y 139.483,Z 963.035,A -85,B 0,C 180,E1 23381.011,E2 23381.011} C_VEL
LIN {X 0,Y 144.053,Z 953.579,A -85,B 0,C 180,E1 23412.148,E2 23412.148} C_VEL
LIN {X 0,Y 171.87,Z 944.375,A -85,B 0,C 180,E1 23428.995,E2 23428.995} C_VEL
LIN {X 0,Y 177.191,Z 942.734,A -85,B 0,C 180,E1 23430.855,E2 23430.855} C_VEL
LIN {X 0,Y 178.144,Z 943.089,A -85,B 0,C 180,E1 23431.798,E2 23431.798} C_VEL
LIN {X 0,Y 155.42,Z 963.52,A -85,B 0,C 180,E1 23440.976,E2 23440.976} C_VEL
LIN {X 0,Y 137.599,Z 977.565,A -85,B 0,C 180,E1 23452.758,E2 23452.758} C_VEL
LIN {X 0,Y 125.186,Z 987.015,A -85,B 0,C 180,E1 23468.726,E2 23468.726} C_VEL
LIN {X 0,Y 120.797,Z 990.547,A -85,B 0,C 180,E1 23485.679,E2 23485.679} C_VEL
LIN {X 0,Y 121.129,Z 990.342,A -85,B 0,C 180,E1 23497.182,E2 23497.182} C_VEL
LIN {X 0,Y 121.769,Z 989.554,A -85,B 0,C 180,E1 23501.583,E2 23501.583} C_VEL
LIN {X 0,Y 121.093,Z 988.375,A -85,B 0,C 180,E1 23507.75,E2 23507.75} C_VEL
LIN {X 0,Y 120.428,Z 985.525,A -85,B 0,C 180,E1 23517.105,E2 23517.105} C_VEL
LIN {X 0,Y 121,Z 985.033,A -85,B 0,C 180,E1 23518.095,E2 23518.095} C_VEL
LIN {X 0,Y 135.133,Z 975.251,A -85,B 0,C 180,E1 23532.244,E2 23532.244} C_VEL
LIN {X 0,Y 156.17,Z 959.083,A -85,B 0,C 180,E1 23543.905,E2 23543.905} C_VEL
LIN {X 0,Y 179.224,Z 938.193,A -85,B 0,C 180,E1 23551.927,E2 23551.927} C_VEL
LIN {X 0,Y 202.437,Z 912.149,A -85,B 0,C 180,E1 23557.607,E2 23557.607} C_VEL
LIN {X 0,Y 212.115,Z 899.108,A -85,B 0,C 180,E1 23559.533,E2 23559.533} C_VEL
LIN {X 0,Y 214.934,Z 887.941,A -85,B 0,C 180,E1 23565.641,E2 23565.641} C_VEL
LIN {X 0,Y 216.366,Z 880.395,A -85,B 0,C 180,E1 23571.946,E2 23571.946} C_VEL
LIN {X 0,Y 218.21,Z 875.658,A -85,B 0,C 180,E1 23579.991,E2 23579.991} C_VEL
LIN {X 0,Y 217.835,Z 881.174,A -85,B 0,C 180,E1 23587.981,E2 23587.981} C_VEL
LIN {X 0,Y 217.422,Z 890.035,A -85,B 0,C 180,E1 23594.457,E2 23594.457} C_VEL
LIN {X 0,Y 216.487,Z 896.921,A -85,B 0,C 180,E1 23597.901,E2 23597.901} C_VEL
LIN {X 0,Y 195.615,Z 925.357,A -85,B 0,C 180,E1 23601.747,E2 23601.747} C_VEL
LIN {X 0,Y 171.301,Z 951.753,A -85,B 0,C 180,E1 23607.884,E2 23607.884} C_VEL
LIN {X 0,Y 147.651,Z 972.772,A -85,B 0,C 180,E1 23616.914,E2 23616.914} C_VEL
LIN {X 0,Y 127.911,Z 988.417,A -85,B 0,C 180,E1 23629.874,E2 23629.874} C_VEL
LIN {X 0,Y 115.809,Z 998.454,A -85,B 0,C 180,E1 23646.906,E2 23646.906} C_VEL
LIN {X 0,Y 112.699,Z 1002.289,A -85,B 0,C 180,E1 23662.278,E2 23662.278} C_VEL
LIN {X 0,Y 112.952,Z 1002.857,A -85,B 0,C 180,E1 23669.999,E2 23669.999} C_VEL
LIN {X 0,Y 113.62,Z 1000.846,A -85,B 0,C 180,E1 23685.456,E2 23685.456} C_VEL
LIN {X 0,Y 122.151,Z 993.083,A -85,B 0,C 180,E1 23703.902,E2 23703.902} C_VEL
LIN {X 0,Y 140.235,Z 978.883,A -85,B 0,C 180,E1 23719.092,E2 23719.092} C_VEL
LIN {X 0,Y 149.684,Z 971.271,A -85,B 0,C 180,E1 23724.018,E2 23724.018} C_VEL
LIN {X 0,Y 150.309,Z 970.207,A -85,B 0,C 180,E1 23724.909,E2 23724.909} C_VEL
LIN {X 0,Y 130.022,Z 965.367,A -85,B 0,C 180,E1 23746.548,E2 23746.548} C_VEL
LIN {X 0,Y 143.688,Z 955.663,A -85,B 0,C 180,E1 23778.442,E2 23778.442} C_VEL
LIN {X 0,Y 168.483,Z 948.343,A -85,B 0,C 180,E1 23791.031,E2 23791.031} C_VEL
LIN {X 0,Y 147.921,Z 965.819,A -85,B 0,C 180,E1 23799.855,E2 23799.855} C_VEL
LIN {X 0,Y 129.552,Z 979.239,A -85,B 0,C 180,E1 23812.153,E2 23812.153} C_VEL
LIN {X 0,Y 117.786,Z 987.425,A -85,B 0,C 180,E1 23827.318,E2 23827.318} C_VEL
LIN {X 0,Y 113.23,Z 990.779,A -85,B 0,C 180,E1 23842.317,E2 23842.317} C_VEL
LIN {X 0,Y 113.038,Z 991.217,A -85,B 0,C 180,E1 23850.001,E2 23850.001} C_VEL
LIN {X 0,Y 116.163,Z 988.508,A -85,B 0,C 180,E1 23869.019,E2 23869.019} C_VEL
LIN {X 0,Y 121,Z 985.033,A -85,B 0,C 180,E1 23878.095,E2 23878.095} C_VEL
LIN {X 0,Y 123.454,Z 981.324,A -85,B 0,C 180,E1 23886.05,E2 23886.05} C_VEL
LIN {X 0,Y 127.779,Z 976.643,A -85,B 0,C 180,E1 23893.529,E2 23893.529} C_VEL
LIN {X 0,Y 149.542,Z 961.139,A -85,B 0,C 180,E1 23905.501,E2 23905.501} C_VEL
LIN {X 0,Y 173.902,Z 940.223,A -85,B 0,C 180,E1 23913.763,E2 23913.763} C_VEL
LIN {X 0,Y 197.79,Z 914.674,A -85,B 0,C 180,E1 23919.373,E2 23919.373} C_VEL
LIN {X 0,Y 206.934,Z 903.012,A -85,B 0,C 180,E1 23921.11,E2 23921.11} C_VEL
LIN {X 0,Y 210.082,Z 893.425,A -85,B 0,C 180,E1 23926.445,E2 23926.445} C_VEL
LIN {X 0,Y 211.711,Z 887.243,A -85,B 0,C 180,E1 23931.768,E2 23931.768} C_VEL
LIN {X 0,Y 212.756,Z 884.094,A -85,B 0,C 180,E1 23935.91,E2 23935.91} C_VEL
LIN {X 0,Y 213.917,Z 882.376,A -85,B 0,C 180,E1 23939.991,E2 23939.991} C_VEL
LIN {X 0,Y 213.306,Z 886.402,A -85,B 0,C 180,E1 23946.404,E2 23946.404} C_VEL
LIN {X 0,Y 212.585,Z 894.921,A -85,B 0,C 180,E1 23953.339,E2 23953.339} C_VEL
LIN {X 0,Y 211.842,Z 899.759,A -85,B 0,C 180,E1 23956.069,E2 23956.069} C_VEL
LIN {X 0,Y 189.538,Z 928.78,A -85,B 0,C 180,E1 23960.175,E2 23960.175} C_VEL
LIN {X 0,Y 164.69,Z 954.034,A -85,B 0,C 180,E1 23966.316,E2 23966.316} C_VEL
LIN {X 0,Y 141.187,Z 973.698,A -85,B 0,C 180,E1 23975.112,E2 23975.112} C_VEL
LIN {X 0,Y 119.743,Z 989.515,A -85,B 0,C 180,E1 23989.319,E2 23989.319} C_VEL
LIN {X 0,Y 108.427,Z 998.038,A -85,B 0,C 180,E1 24005.232,E2 24005.232} C_VEL
LIN {X 0,Y 104.816,Z 1001.879,A -85,B 0,C 180,E1 24021.693,E2 24021.693} C_VEL
LIN {X 0,Y 105.048,Z 1002.45,A -85,B 0,C 180,E1 24029.999,E2 24029.999} C_VEL
LIN {X 0,Y 105.912,Z 1000.433,A -85,B 0,C 180,E1 24046.612,E2 24046.612} C_VEL
LIN {X 0,Y 115.499,Z 992.666,A -85,B 0,C 180,E1 24066.149,E2 24066.149} C_VEL
LIN {X 0,Y 135.074,Z 978.469,A -85,B 0,C 180,E1 24081.687,E2 24081.687} C_VEL
LIN {X 0,Y 139.681,Z 975.03,A -85,B 0,C 180,E1 24084.124,E2 24084.124} C_VEL
LIN {X 0,Y 140.603,Z 973.344,A -85,B 0,C 180,E1 24085.736,E2 24085.736} C_VEL
LIN {X 0,Y 123.226,Z 969.181,A -85,B 0,C 180,E1 24105.791,E2 24105.791} C_VEL
LIN {X 0,Y 137.174,Z 959.815,A -85,B 0,C 180,E1 24139.351,E2 24139.351} C_VEL
LIN {X 0,Y 157.879,Z 954.093,A -85,B 0,C 180,E1 24150.525,E2 24150.525} C_VEL
LIN {X 0,Y 155.956,Z 956.239,A -85,B 0,C 180,E1 24151.91,E2 24151.91} C_VEL
LIN {X 0,Y 134.143,Z 972.441,A -85,B 0,C 180,E1 24162.143,E2 24162.143} C_VEL
LIN {X 0,Y 118.226,Z 982.919,A -85,B 0,C 180,E1 24174.81,E2 24174.81} C_VEL
LIN {X 0,Y 107.211,Z 989.921,A -85,B 0,C 180,E1 24193.595,E2 24193.595} C_VEL
LIN {X 0,Y 105.16,Z 991.623,A -85,B 0,C 180,E1 24210.001,E2 24210.001} C_VEL
LIN {X 0,Y 107.217,Z 989.878,A -85,B 0,C 180,E1 24226.407,E2 24226.407} C_VEL
LIN {X 0,Y 118.264,Z 982.827,A -85,B 0,C 180,E1 24245.18,E2 24245.18} C_VEL
LIN {X 0,Y 127.779,Z 976.643,A -85,B 0,C 180,E1 24253.529,E2 24253.529} C_VEL
LIN {X 0,Y 133.742,Z 971.087,A -85,B 0,C 180,E1 24260.34,E2 24260.34} C_VEL
LIN {X 0,Y 141.014,Z 964.497,A -85,B 0,C 180,E1 24266.411,E2 24266.411} C_VEL
LIN {X 0,Y 166.823,Z 944.056,A -85,B 0,C 180,E1 24275.179,E2 24275.179} C_VEL
LIN {X 0,Y 192.166,Z 918.473,A -85,B 0,C 180,E1 24280.997,E2 24280.997} C_VEL
LIN {X 0,Y 202.794,Z 905.446,A -85,B 0,C 180,E1 24283.166,E2 24283.166} C_VEL
LIN {X 0,Y 206.096,Z 896.177,A -85,B 0,C 180,E1 24289.408,E2 24289.408} C_VEL
LIN {X 0,Y 208.101,Z 890.755,A -85,B 0,C 180,E1 24295.818,E2 24295.818} C_VEL
LIN {X 0,Y 209.399,Z 888.959,A -85,B 0,C 180,E1 24299.991,E2 24299.991} C_VEL
LIN {X 0,Y 208.614,Z 893.111,A -85,B 0,C 180,E1 24306.548,E2 24306.548} C_VEL
LIN {X 0,Y 207.574,Z 900.432,A -85,B 0,C 180,E1 24312.63,E2 24312.63} C_VEL
LIN {X 0,Y 206.643,Z 903.962,A -85,B 0,C 180,E1 24314.568,E2 24314.568} C_VEL
LIN {X 0,Y 183.606,Z 931.903,A -85,B 0,C 180,E1 24318.495,E2 24318.495} C_VEL
LIN {X 0,Y 158.207,Z 956.304,A -85,B 0,C 180,E1 24324.606,E2 24324.606} C_VEL
LIN {X 0,Y 132.711,Z 976.168,A -85,B 0,C 180,E1 24334.192,E2 24334.192} C_VEL
LIN {X 0,Y 112.53,Z 989.835,A -85,B 0,C 180,E1 24347.719,E2 24347.719} C_VEL
LIN {X 0,Y 99.295,Z 999.079,A -85,B 0,C 180,E1 24368.211,E2 24368.211} C_VEL
LIN {X 0,Y 96.927,Z 1001.467,A -85,B 0,C 180,E1 24381.012,E2 24381.012} C_VEL
LIN {X 0,Y 97.128,Z 1002.042,A -85,B 0,C 180,E1 24389.999,E2 24389.999} C_VEL
LIN {X 0,Y 98.239,Z 1000.02,A -85,B 0,C 180,E1 24407.952,E2 24407.952} C_VEL
LIN {X 0,Y 109.071,Z 992.25,A -85,B 0,C 180,E1 24428.657,E2 24428.657} C_VEL
LIN {X 0,Y 130.198,Z 978.054,A -85,B 0,C 180,E1 24444.491,E2 24444.491} C_VEL
LIN {X 0,Y 131.838,Z 976.448,A -85,B 0,C 180,E1 24445.993,E2 24445.993} C_VEL
LIN {X 0,Y 115.035,Z 971.182,A -85,B 0,C 180,E1 24472.454,E2 24472.454} C_VEL
LIN {X 0,Y 147.572,Z 959.851,A -85,B 0,C 180,E1 24510.877,E2 24510.877} C_VEL
LIN {X 0,Y 123.669,Z 976.212,A -85,B 0,C 180,E1 24522.729,E2 24522.729} C_VEL
LIN {X 0,Y 106.866,Z 986.158,A -85,B 0,C 180,E1 24538.251,E2 24538.251} C_VEL
LIN {X 0,Y 99.611,Z 990.33,A -85,B 0,C 180,E1 24552.303,E2 24552.303} C_VEL
LIN {X 0,Y 97.259,Z 992.03,A -85,B 0,C 180,E1 24570.001,E2 24570.001} C_VEL
LIN {X 0,Y 99.617,Z 990.287,A -85,B 0,C 180,E1 24587.698,E2 24587.698} C_VEL
LIN {X 0,Y 111.825,Z 983.239,A -85,B 0,C 180,E1 24607.54,E2 24607.54} C_VEL
LIN {X 0,Y 133.181,Z 969.907,A -85,B 0,C 180,E1 24622.733,E2 24622.733} C_VEL
LIN {X 0,Y 141.014,Z 964.497,A -85,B 0,C 180,E1 24626.411,E2 24626.411} C_VEL
LIN {X 0,Y 149.451,Z 957.102,A -85,B 0,C 180,E1 24631.746,E2 24631.746} C_VEL
LIN {X 0,Y 158.538,Z 948.688,A -85,B 0,C 180,E1 24636.365,E2 24636.365} C_VEL
LIN {X 0,Y 183.063,Z 926.044,A -85,B 0,C 180,E1 24642.02,E2 24642.02} C_VEL
LIN {X 0,Y 197.695,Z 909.608,A -85,B 0,C 180,E1 24644.627,E2 24644.627} C_VEL
LIN {X 0,Y 201.175,Z 901.75,A -85,B 0,C 180,E1 24650.139,E2 24650.139} C_VEL
LIN {X 0,Y 203.191,Z 897.274,A -85,B 0,C 180,E1 24655.717,E2 24655.717} C_VEL
LIN {X 0,Y 204.643,Z 895.365,A -85,B 0,C 180,E1 24659.99,E2 24659.99} C_VEL
LIN {X 0,Y 203.562,Z 900.422,A -85,B 0,C 180,E1 24667.469,E2 24667.469} C_VEL
LIN {X 0,Y 201.846,Z 907.416,A -85,B 0,C 180,E1 24672.794,E2 24672.794} C_VEL
LIN {X 0,Y 177.839,Z 935.024,A -85,B 0,C 180,E1 24676.701,E2 24676.701} C_VEL
LIN {X 0,Y 151.886,Z 958.445,A -85,B 0,C 180,E1 24682.763,E2 24682.763} C_VEL
LIN {X 0,Y 125.613,Z 977.528,A -85,B 0,C 180,E1 24692.459,E2 24692.459} C_VEL
LIN {X 0,Y 105.573,Z 990.074,A -85,B 0,C 180,E1 24705.784,E2 24705.784} C_VEL
LIN {X 0,Y 91.735,Z 998.771,A -85,B 0,C 180,E1 24726.739,E2 24726.739} C_VEL
LIN {X 0,Y 89.059,Z 1001.057,A -85,B 0,C 180,E1 24740.21,E2 24740.21} C_VEL
LIN {X 0,Y 89.228,Z 1001.635,A -85,B 0,C 180,E1 24749.999,E2 24749.999} C_VEL
LIN {X 0,Y 90.653,Z 999.608,A -85,B 0,C 180,E1 24769.513,E2 24769.513} C_VEL
LIN {X 0,Y 102.424,Z 992.08,A -85,B 0,C 180,E1 24791.008,E2 24791.008} C_VEL
LIN {X 0,Y 122.812,Z 979.333,A -85,B 0,C 180,E1 24806.423,E2 24806.423} C_VEL
LIN {X 0,Y 108.617,Z 972.985,A -85,B 0,C 180,E1 24840.018,E2 24840.018} C_VEL
LIN {X 0,Y 136.986,Z 964.484,A -85,B 0,C 180,E1 24869.841,E2 24869.841} C_VEL
LIN {X 0,Y 133.794,Z 967.046,A -85,B 0,C 180,E1 24871.927,E2 24871.927} C_VEL
LIN {X 0,Y 111.576,Z 980.47,A -85,B 0,C 180,E1 24884.569,E2 24884.569} C_VEL
LIN {X 0,Y 96.169,Z 988.655,A -85,B 0,C 180,E1 24901.816,E2 24901.816} C_VEL
LIN {X 0,Y 89.769,Z 992.001,A -85,B 0,C 180,E1 24920.291,E2 24920.291} C_VEL
LIN {X 0,Y 89.368,Z 992.437,A -85,B 0,C 180,E1 24930.001,E2 24930.001} C_VEL
LIN {X 0,Y 92.076,Z 990.697,A -85,B 0,C 180,E1 24949.202,E2 24949.202} C_VEL
LIN {X 0,Y 105.584,Z 983.652,A -85,B 0,C 180,E1 24970.19,E2 24970.19} C_VEL
LIN {X 0,Y 128.489,Z 970.319,A -85,B 0,C 180,E1 24985.577,E2 24985.577} C_VEL
LIN {X 0,Y 154.32,Z 952.102,A -85,B 0,C 180,E1 24995.172,E2 24995.172} C_VEL
LIN {X 0,Y 158.538,Z 948.688,A -85,B 0,C 180,E1 24996.365,E2 24996.365} C_VEL
LIN {X 0,Y 168.139,Z 939.526,A -85,B 0,C 180,E1 25000.399,E2 25000.399} C_VEL
LIN {X 0,Y 177.833,Z 929.426,A -85,B 0,C 180,E1 25003.881,E2 25003.881} C_VEL
LIN {X 0,Y 192.778,Z 913.527,A -85,B 0,C 180,E1 25006.428,E2 25006.428} C_VEL
LIN {X 0,Y 195.586,Z 908.422,A -85,B 0,C 180,E1 25009.854,E2 25009.854} C_VEL
LIN {X 0,Y 198.053,Z 903.61,A -85,B 0,C 180,E1 25015.606,E2 25015.606} C_VEL
LIN {X 0,Y 199.708,Z 901.679,A -85,B 0,C 180,E1 25019.99,E2 25019.99} C_VEL
LIN {X 0,Y 198.399,Z 906.409,A -85,B 0,C 180,E1 25027.201,E2 25027.201} C_VEL
LIN {X 0,Y 197.448,Z 910.218,A -85,B 0,C 180,E1 25030.507,E2 25030.507} C_VEL
LIN {X 0,Y 193.763,Z 914.993,A -85,B 0,C 180,E1 25031.426,E2 25031.426} C_VEL
LIN {X 0,Y 169.098,Z 940.887,A -85,B 0,C 180,E1 25035.38,E2 25035.38} C_VEL
LIN {X 0,Y 142.143,Z 963.203,A -85,B 0,C 180,E1 25041.771,E2 25041.771} C_VEL
LIN {X 0,Y 114.245,Z 981.487,A -85,B 0,C 180,E1 25052.766,E2 25052.766} C_VEL
LIN {X 0,Y 93.085,Z 993.368,A -85,B 0,C 180,E1 25069.409,E2 25069.409} C_VEL
LIN {X 0,Y 83.097,Z 999.165,A -85,B 0,C 180,E1 25088.627,E2 25088.627} C_VEL
LIN {X 0,Y 81.302,Z 1001.227,A -85,B 0,C 180,E1 25109.998,E2 25109.998} C_VEL
LIN {X 0,Y 83.12,Z 999.194,A -85,B 0,C 180,E1 25131.364,E2 25131.364} C_VEL
LIN {X 0,Y 96.138,Z 991.819,A -85,B 0,C 180,E1 25153.868,E2 25153.868} C_VEL
LIN {X 0,Y 110.648,Z 983.745,A -85,B 0,C 180,E1 25165.186,E2 25165.186} C_VEL
LIN {X 0,Y 112.935,Z 981.804,A -85,B 0,C 180,E1 25167.592,E2 25167.592} C_VEL
LIN {X 0,Y 104.493,Z 974.598,A -85,B 0,C 180,E1 25208.35,E2 25208.35} C_VEL
LIN {X 0,Y 127.216,Z 968.745,A -85,B 0,C 180,E1 25229.299,E2 25229.299} C_VEL
LIN {X 0,Y 121.311,Z 972.573,A -85,B 0,C 180,E1 25232.6,E2 25232.6} C_VEL
LIN {X 0,Y 99.563,Z 984.152,A -85,B 0,C 180,E1 25246.818,E2 25246.818} C_VEL
LIN {X 0,Y 84.601,Z 991.148,A -85,B 0,C 180,E1 25269.028,E2 25269.028} C_VEL
LIN {X 0,Y 81.466,Z 992.844,A -85,B 0,C 180,E1 25290.002,E2 25290.002} C_VEL
LIN {X 0,Y 84.608,Z 991.107,A -85,B 0,C 180,E1 25310.973,E2 25310.973} C_VEL
LIN {X 0,Y 99.612,Z 984.064,A -85,B 0,C 180,E1 25333.158,E2 25333.158} C_VEL
LIN {X 0,Y 124.129,Z 970.732,A -85,B 0,C 180,E1 25348.634,E2 25348.634} C_VEL
LIN {X 0,Y 151.135,Z 952.512,A -85,B 0,C 180,E1 25357.925,E2 25357.925} C_VEL
LIN {X 0,Y 177.833,Z 929.426,A -85,B 0,C 180,E1 25363.881,E2 25363.881} C_VEL
LIN {X 0,Y 184.827,Z 921.824,A -85,B 0,C 180,E1 25365.892,E2 25365.892} C_VEL
LIN {X 0,Y 189.17,Z 915.88,A -85,B 0,C 180,E1 25368.815,E2 25368.815} C_VEL
LIN {X 0,Y 191.672,Z 911.45,A -85,B 0,C 180,E1 25373.185,E2 25373.185} C_VEL
LIN {X 0,Y 194.585,Z 907.862,A -85,B 0,C 180,E1 25379.99,E2 25379.99} C_VEL
LIN {X 0,Y 192.916,Z 912.781,A -85,B 0,C 180,E1 25387.407,E2 25387.407} C_VEL
LIN {X 0,Y 192.357,Z 914.534,A -85,B 0,C 180,E1 25389.047,E2 25389.047} C_VEL
LIN {X 0,Y 165.167,Z 942.3,A -85,B 0,C 180,E1 25393.061,E2 25393.061} C_VEL
LIN {X 0,Y 136.627,Z 964.618,A -85,B 0,C 180,E1 25399.402,E2 25399.402} C_VEL
LIN {X 0,Y 108.052,Z 982.188,A -85,B 0,C 180,E1 25410.211,E2 25410.211} C_VEL
LIN {X 0,Y 87.083,Z 992.95,A -85,B 0,C 180,E1 25425.933,E2 25425.933} C_VEL
LIN {X 0,Y 75.661,Z 998.751,A -85,B 0,C 180,E1 25446.405,E2 25446.405} C_VEL
LIN {X 0,Y 73.389,Z 1000.819,A -85,B 0,C 180,E1 25469.998,E2 25469.998} C_VEL
LIN {X 0,Y 75.684,Z 998.781,A -85,B 0,C 180,E1 25493.583,E2 25493.583} C_VEL
LIN {X 0,Y 92.03,Z 990.658,A -85,B 0,C 180,E1 25518.877,E2 25518.877} C_VEL
LIN {X 0,Y 102.7,Z 985.151,A -85,B 0,C 180,E1 25526.735,E2 25526.735} C_VEL
LIN {X 0,Y 103.876,Z 984.196,A -85,B 0,C 180,E1 25528.261,E2 25528.261} C_VEL
LIN {X 0,Y 97.199,Z 977.662,A -85,B 0,C 180,E1 25568.981,E2 25568.981} C_VEL
LIN {X 0,Y 116.573,Z 972.955,A -85,B 0,C 180,E1 25588.493,E2 25588.493} C_VEL
LIN {X 0,Y 111.545,Z 975.971,A -85,B 0,C 180,E1 25591.968,E2 25591.968} C_VEL
LIN {X 0,Y 89.643,Z 986.403,A -85,B 0,C 180,E1 25607.501,E2 25607.501} C_VEL
LIN {X 0,Y 77.233,Z 991.557,A -85,B 0,C 180,E1 25626.917,E2 25626.917} C_VEL
LIN {X 0,Y 73.568,Z 993.25,A -85,B 0,C 180,E1 25650.002,E2 25650.002} C_VEL
LIN {X 0,Y 77.24,Z 991.516,A -85,B 0,C 180,E1 25673.084,E2 25673.084} C_VEL
LIN {X 0,Y 93.95,Z 984.475,A -85,B 0,C 180,E1 25696.489,E2 25696.489} C_VEL
LIN {X 0,Y 120.156,Z 971.144,A -85,B 0,C 180,E1 25711.896,E2 25711.896} C_VEL
LIN {X 0,Y 148.312,Z 952.924,A -85,B 0,C 180,E1 25720.792,E2 25720.792} C_VEL
LIN {X 0,Y 175.326,Z 930.29,A -85,B 0,C 180,E1 25726.3,E2 25726.3} C_VEL
LIN {X 0,Y 189.043,Z 916.095,A -85,B 0,C 180,E1 25728.64,E2 25728.64} C_VEL
LIN {X 0,Y 189.17,Z 915.88,A -85,B 0,C 180,E1 25728.815,E2 25728.815} C_VEL
LIN {X 0,Y 189.625,Z 913.933,A -85,B 0,C 180,E1 25732.717,E2 25732.717} C_VEL
LIN {X 0,Y 188.959,Z 914.035,A -85,B 0,C 180,E1 25739.553,E2 25739.553} C_VEL
LIN {X 0,Y 188.229,Z 916.346,A -85,B 0,C 180,E1 25744.603,E2 25744.603} C_VEL
LIN {X 0,Y 187.119,Z 918.864,A -85,B 0,C 180,E1 25747.173,E2 25747.173} C_VEL
LIN {X 0,Y 159.551,Z 945.195,A -85,B 0,C 180,E1 25750.928,E2 25750.928} C_VEL
LIN {X 0,Y 130.727,Z 966.46,A -85,B 0,C 180,E1 25757.023,E2 25757.023} C_VEL
LIN {X 0,Y 102.229,Z 982.818,A -85,B 0,C 180,E1 25767.293,E2 25767.293} C_VEL
LIN {X 0,Y 77.308,Z 994.335,A -85,B 0,C 180,E1 25786.724,E2 25786.724} C_VEL
LIN {X 0,Y 68.346,Z 998.335,A -85,B 0,C 180,E1 25803.698,E2 25803.698} C_VEL
LIN {X 0,Y 65.455,Z 1000.411,A -85,B 0,C 180,E1 25829.998,E2 25829.998} C_VEL
LIN {X 0,Y 69.44,Z 997.901,A -85,B 0,C 180,E1 25859.351,E2 25859.351} C_VEL
LIN {X 0,Y 88.998,Z 989.238,A -85,B 0,C 180,E1 25884.567,E2 25884.567} C_VEL
LIN {X 0,Y 93.185,Z 987.318,A -85,B 0,C 180,E1 25887.518,E2 25887.518} C_VEL
LIN {X 0,Y 94.309,Z 986.301,A -85,B 0,C 180,E1 25889.606,E2 25889.606} C_VEL
LIN {X 0,Y 95.768,Z 978.957,A -85,B 0,C 180,E1 25938.454,E2 25938.454} C_VEL
LIN {X 0,Y 106.645,Z 976.652,A -85,B 0,C 180,E1 25948.121,E2 25948.121} C_VEL
LIN {X 0,Y 91.04,Z 983.908,A -85,B 0,C 180,E1 25957.819,E2 25957.819} C_VEL
LIN {X 0,Y 72.673,Z 991.027,A -85,B 0,C 180,E1 25978.612,E2 25978.612} C_VEL
LIN {X 0,Y 65.665,Z 993.657,A -85,B 0,C 180,E1 26010.002,E2 26010.002} C_VEL
LIN {X 0,Y 69.992,Z 991.926,A -85,B 0,C 180,E1 26035.638,E2 26035.638} C_VEL
LIN {X 0,Y 88.638,Z 984.887,A -85,B 0,C 180,E1 26060.238,E2 26060.238} C_VEL
LIN {X 0,Y 116.597,Z 971.557,A -85,B 0,C 180,E1 26075.371,E2 26075.371} C_VEL
LIN {X 0,Y 145.88,Z 953.333,A -85,B 0,C 180,E1 26083.755,E2 26083.755} C_VEL
LIN {X 0,Y 173.61,Z 930.698,A -85,B 0,C 180,E1 26088.857,E2 26088.857} C_VEL
LIN {X 0,Y 184.427,Z 919.891,A -85,B 0,C 180,E1 26090.539,E2 26090.539} C_VEL
LIN {X 0,Y 187.186,Z 915.96,A -85,B 0,C 180,E1 26095.35,E2 26095.35} C_VEL
LIN {X 0,Y 188.959,Z 914.035,A -85,B 0,C 180,E1 26099.553,E2 26099.553} C_VEL
LIN {X 0,Y 188.337,Z 915.247,A -85,B 0,C 180,E1 26101.866,E2 26101.866} C_VEL
LIN {X 0,Y 183.743,Z 920.946,A -85,B 0,C 180,E1 26104.513,E2 26104.513} C_VEL
LIN {X 0,Y 179.772,Z 925.25,A -85,B 0,C 180,E1 26105.381,E2 26105.381} C_VEL
LIN {X 0,Y 151.425,Z 950.196,A -85,B 0,C 180,E1 26109.101,E2 26109.101} C_VEL
LIN {X 0,Y 121.64,Z 970.221,A -85,B 0,C 180,E1 26115.271,E2 26115.271} C_VEL
LIN {X 0,Y 92.687,Z 985.178,A -85,B 0,C 180,E1 26126.041,E2 26126.041} C_VEL
LIN {X 0,Y 67.482,Z 995.536,A -85,B 0,C 180,E1 26147.69,E2 26147.69} C_VEL
LIN {X 0,Y 57.823,Z 999.41,A -85,B 0,C 180,E1 26174.818,E2 26174.818} C_VEL
LIN {X 0,Y 57.521,Z 1000.002,A -85,B 0,C 180,E1 26189.998,E2 26189.998} C_VEL
LIN {X 0,Y 61.247,Z 997.951,A -85,B 0,C 180,E1 26219.629,E2 26219.629} C_VEL
LIN {X 0,Y 82.528,Z 989.705,A -85,B 0,C 180,E1 26247.636,E2 26247.636} C_VEL
LIN {X 0,Y 84.197,Z 988.973,A -85,B 0,C 180,E1 26248.817,E2 26248.817} C_VEL
LIN {X 0,Y 84.908,Z 988.138,A -85,B 0,C 180,E1 26251.129,E2 26251.129} C_VEL
LIN {X 0,Y 94.07,Z 980.528,A -85,B 0,C 180,E1 26305.495,E2 26305.495} C_VEL
LIN {X 0,Y 96.246,Z 980.134,A -85,B 0,C 180,E1 26307.347,E2 26307.347} C_VEL
LIN {X 0,Y 73.903,Z 988.848,A -85,B 0,C 180,E1 26324.19,E2 26324.19} C_VEL
LIN {X 0,Y 58.764,Z 993.632,A -85,B 0,C 180,E1 26355.071,E2 26355.071} C_VEL
LIN {X 0,Y 57.778,Z 994.064,A -85,B 0,C 180,E1 26370.002,E2 26370.002} C_VEL
LIN {X 0,Y 65.974,Z 991.394,A -85,B 0,C 180,E1 26404.924,E2 26404.924} C_VEL
LIN {X 0,Y 89.196,Z 983.116,A -85,B 0,C 180,E1 26428.078,E2 26428.078} C_VEL
LIN {X 0,Y 118.853,Z 969.19,A -85,B 0,C 180,E1 26440.726,E2 26440.726} C_VEL
LIN {X 0,Y 148.586,Z 950.363,A -85,B 0,C 180,E1 26447.729,E2 26447.729} C_VEL
LIN {X 0,Y 176.296,Z 927.255,A -85,B 0,C 180,E1 26451.997,E2 26451.997} C_VEL
LIN {X 0,Y 179.153,Z 924.549,A -85,B 0,C 180,E1 26452.358,E2 26452.358} C_VEL
LIN {X 0,Y 181.366,Z 921.859,A -85,B 0,C 180,E1 26455.201,E2 26455.201} C_VEL
LIN {X 0,Y 183.657,Z 919.684,A -85,B 0,C 180,E1 26459.989,E2 26459.989} C_VEL
LIN {X 0,Y 182.39,Z 922.474,A -85,B 0,C 180,E1 26465.01,E2 26465.01} C_VEL
LIN {X 0,Y 179.772,Z 925.25,A -85,B 0,C 180,E1 26465.381,E2 26465.381} C_VEL
LIN {X 0,Y 166.709,Z 936.993,A -85,B 0,C 180,E1 26465.448,E2 26465.448} C_VEL
LIN {X 0,Y 154.65,Z 946.509,A -85,B 0,C 180,E1 26465.505,E2 26465.505} C_VEL
LIN {X 0,Y 152.977,Z 947.817,A -85,B 0,C 180,E1 26465.696,E2 26465.696} C_VEL
LIN {X 0,Y 123.294,Z 967.818,A -85,B 0,C 180,E1 26470.751,E2 26470.751} C_VEL
LIN {X 0,Y 92.62,Z 983.378,A -85,B 0,C 180,E1 26479.949,E2 26479.949} C_VEL
LIN {X 0,Y 66.425,Z 993.499,A -85,B 0,C 180,E1 26497.077,E2 26497.077} C_VEL
LIN {X 0,Y 53.925,Z 997.649,A -85,B 0,C 180,E1 26517.316,E2 26517.316} C_VEL
LIN {X 0,Y 49.581,Z 999.593,A -85,B 0,C 180,E1 26549.997,E2 26549.997} C_VEL
LIN {X 0,Y 54.382,Z 997.536,A -85,B 0,C 180,E1 26583.835,E2 26583.835} C_VEL
LIN {X 0,Y 74.812,Z 990.614,A -85,B 0,C 180,E1 26610.144,E2 26610.144} C_VEL
LIN {X 0,Y 76.158,Z 989.94,A -85,B 0,C 180,E1 26611.996,E2 26611.996} C_VEL
LIN {X 0,Y 81.627,Z 984.063,A -85,B 0,C 180,E1 26661.964,E2 26661.964} C_VEL
LIN {X 0,Y 85.171,Z 983.627,A -85,B 0,C 180,E1 26667.274,E2 26667.274} C_VEL
LIN {X 0,Y 61.834,Z 991.232,A -85,B 0,C 180,E1 26687.315,E2 26687.315} C_VEL
LIN {X 0,Y 51.143,Z 994.041,A -85,B 0,C 180,E1 26712.782,E2 26712.782} C_VEL
LIN {X 0,Y 49.873,Z 994.471,A -85,B 0,C 180,E1 26730.003,E2 26730.003} C_VEL
LIN {X 0,Y 56.079,Z 992.746,A -85,B 0,C 180,E1 26762.685,E2 26762.685} C_VEL
LIN {X 0,Y 79.361,Z 985.712,A -85,B 0,C 180,E1 26789.156,E2 26789.156} C_VEL
LIN {X 0,Y 110.883,Z 972.38,A -85,B 0,C 180,E1 26802.913,E2 26802.913} C_VEL
LIN {X 0,Y 141.631,Z 954.553,A -85,B 0,C 180,E1 26809.842,E2 26809.842} C_VEL
LIN {X 0,Y 171.758,Z 931.035,A -85,B 0,C 180,E1 26814.148,E2 26814.148} C_VEL
LIN {X 0,Y 174.572,Z 928.403,A -85,B 0,C 180,E1 26814.477,E2 26814.477} C_VEL
LIN {X 0,Y 177.942,Z 925.412,A -85,B 0,C 180,E1 26819.989,E2 26819.989} C_VEL
LIN {X 0,Y 177.415,Z 926.432,A -85,B 0,C 180,E1 26822.434,E2 26822.434} C_VEL
LIN {X 0,Y 175.061,Z 928.819,A -85,B 0,C 180,E1 26823.207,E2 26823.207} C_VEL
LIN {X 0,Y 152.977,Z 947.817,A -85,B 0,C 180,E1 26825.696,E2 26825.696} C_VEL
LIN {X 0,Y 138.567,Z 957.74,A -85,B 0,C 180,E1 26826.149,E2 26826.149} C_VEL
LIN {X 0,Y 123.477,Z 966.583,A -85,B 0,C 180,E1 26826.756,E2 26826.756} C_VEL
LIN {X 0,Y 90.173,Z 982.959,A -85,B 0,C 180,E1 26835.093,E2 26835.093} C_VEL
LIN {X 0,Y 61.671,Z 993.142,A -85,B 0,C 180,E1 26851.269,E2 26851.269} C_VEL
LIN {X 0,Y 42.581,Z 998.585,A -85,B 0,C 180,E1 26889.168,E2 26889.168} C_VEL
LIN {X 0,Y 41.636,Z 999.184,A -85,B 0,C 180,E1 26909.997,E2 26909.997} C_VEL
LIN {X 0,Y 47.881,Z 997.12,A -85,B 0,C 180,E1 26949.226,E2 26949.226} C_VEL
LIN {X 0,Y 67.268,Z 991.471,A -85,B 0,C 180,E1 26973.28,E2 26973.28} C_VEL
LIN {X 0,Y 75.145,Z 986.249,A -85,B 0,C 180,E1 27024.919,E2 27024.919} C_VEL
LIN {X 0,Y 69.499,Z 988.046,A -85,B 0,C 180,E1 27029.378,E2 27029.378} C_VEL
LIN {X 0,Y 49.551,Z 993.194,A -85,B 0,C 180,E1 27052.332,E2 27052.332} C_VEL
LIN {X 0,Y 41.985,Z 994.877,A -85,B 0,C 180,E1 27090.003,E2 27090.003} C_VEL
LIN {X 0,Y 49.565,Z 993.156,A -85,B 0,C 180,E1 27127.662,E2 27127.662} C_VEL
LIN {X 0,Y 75.579,Z 986.123,A -85,B 0,C 180,E1 27154.36,E2 27154.36} C_VEL
LIN {X 0,Y 108.803,Z 972.792,A -85,B 0,C 180,E1 27166.941,E2 27166.941} C_VEL
LIN {X 0,Y 140.008,Z 955.242,A -85,B 0,C 180,E1 27172.987,E2 27172.987} C_VEL
LIN {X 0,Y 168.364,Z 933.86,A -85,B 0,C 180,E1 27176.531,E2 27176.531} C_VEL
LIN {X 0,Y 170.577,Z 931.957,A -85,B 0,C 180,E1 27177.338,E2 27177.338} C_VEL
LIN {X 0,Y 171.962,Z 930.983,A -85,B 0,C 180,E1 27180.399,E2 27180.399} C_VEL
LIN {X 0,Y 169.672,Z 933.186,A -85,B 0,C 180,E1 27180.991,E2 27180.991} C_VEL
LIN {X 0,Y 138.55,Z 957.181,A -85,B 0,C 180,E1 27184.388,E2 27184.388} C_VEL
LIN {X 0,Y 123.477,Z 966.583,A -85,B 0,C 180,E1 27186.756,E2 27186.756} C_VEL
LIN {X 0,Y 107.879,Z 974.465,A -85,B 0,C 180,E1 27187.636,E2 27187.636} C_VEL
LIN {X 0,Y 91.89,Z 981.179,A -85,B 0,C 180,E1 27189.018,E2 27189.018} C_VEL
LIN {X 0,Y 57.421,Z 992.846,A -85,B 0,C 180,E1 27204.732,E2 27204.732} C_VEL
LIN {X 0,Y 35.2,Z 998.172,A -85,B 0,C 180,E1 27244.52,E2 27244.52} C_VEL
LIN {X 0,Y 33.688,Z 998.774,A -85,B 0,C 180,E1 27269.996,E2 27269.996} C_VEL
LIN {X 0,Y 41.944,Z 996.706,A -85,B 0,C 180,E1 27316.211,E2 27316.211} C_VEL
LIN {X 0,Y 57.56,Z 992.87,A -85,B 0,C 180,E1 27335.325,E2 27335.325} C_VEL
LIN {X 0,Y 64.394,Z 988.814,A -85,B 0,C 180,E1 27382.7,E2 27382.7} C_VEL
LIN {X 0,Y 59.71,Z 990.081,A -85,B 0,C 180,E1 27387.443,E2 27387.443} C_VEL
LIN {X 0,Y 43.52,Z 993.604,A -85,B 0,C 180,E1 27405.912,E2 27405.912} C_VEL
LIN {X 0,Y 34.078,Z 995.284,A -85,B 0,C 180,E1 27450.004,E2 27450.004} C_VEL
LIN {X 0,Y 47.963,Z 992.715,A -85,B 0,C 180,E1 27500.8,E2 27500.8} C_VEL
LIN {X 0,Y 79.165,Z 984.353,A -85,B 0,C 180,E1 27523.002,E2 27523.002} C_VEL
LIN {X 0,Y 113.534,Z 970.265,A -85,B 0,C 180,E1 27532.319,E2 27532.319} C_VEL
LIN {X 0,Y 145.565,Z 951.472,A -85,B 0,C 180,E1 27537.016,E2 27537.016} C_VEL
LIN {X 0,Y 162.563,Z 938.849,A -85,B 0,C 180,E1 27538.785,E2 27538.785} C_VEL
LIN {X 0,Y 130.667,Z 961.529,A -85,B 0,C 180,E1 27541.935,E2 27541.935} C_VEL
LIN {X 0,Y 99.198,Z 977.995,A -85,B 0,C 180,E1 27547.19,E2 27547.19} C_VEL
LIN {X 0,Y 91.89,Z 981.179,A -85,B 0,C 180,E1 27549.018,E2 27549.018} C_VEL
LIN {X 0,Y 75.516,Z 986.782,A -85,B 0,C 180,E1 27551.121,E2 27551.121} C_VEL
LIN {X 0,Y 59,Z 991.285,A -85,B 0,C 180,E1 27554.4,E2 27554.4} C_VEL
LIN {X 0,Y 36.81,Z 996.256,A -85,B 0,C 180,E1 27574.643,E2 27574.643} C_VEL
LIN {X 0,Y 25.741,Z 998.365,A -85,B 0,C 180,E1 27629.995,E2 27629.995} C_VEL
LIN {X 0,Y 36.818,Z 996.29,A -85,B 0,C 180,E1 27685.326,E2 27685.326} C_VEL
LIN {X 0,Y 48.69,Z 993.914,A -85,B 0,C 180,E1 27698.882,E2 27698.882} C_VEL
LIN {X 0,Y 53.696,Z 991.065,A -85,B 0,C 180,E1 27739.638,E2 27739.638} C_VEL
LIN {X 0,Y 50.006,Z 991.937,A -85,B 0,C 180,E1 27744.727,E2 27744.727} C_VEL
LIN {X 0,Y 29.277,Z 995.265,A -85,B 0,C 180,E1 27778.864,E2 27778.864} C_VEL
LIN {X 0,Y 26.17,Z 995.692,A -85,B 0,C 180,E1 27810.005,E2 27810.005} C_VEL
LIN {X 0,Y 43.361,Z 993.127,A -85,B 0,C 180,E1 27869.001,E2 27869.001} C_VEL
LIN {X 0,Y 77.208,Z 984.765,A -85,B 0,C 180,E1 27888.683,E2 27888.683} C_VEL
LIN {X 0,Y 112.743,Z 970.677,A -85,B 0,C 180,E1 27896.36,E2 27896.36} C_VEL
LIN {X 0,Y 128.934,Z 962.104,A -85,B 0,C 180,E1 27898.545,E2 27898.545} C_VEL
LIN {X 0,Y 94.779,Z 979.152,A -85,B 0,C 180,E1 27903.181,E2 27903.181} C_VEL
LIN {X 0,Y 59,Z 991.285,A -85,B 0,C 180,E1 27914.4,E2 27914.4} C_VEL
LIN {X 0,Y 42.55,Z 994.595,A -85,B 0,C 180,E1 27920.201,E2 27920.201} C_VEL
LIN {X 0,Y 26.648,Z 996.672,A -85,B 0,C 180,E1 27932.628,E2 27932.628} C_VEL
LIN {X 0,Y 17.784,Z 997.955,A -85,B 0,C 180,E1 27989.993,E2 27989.993} C_VEL
LIN {X 0,Y 36.781,Z 995.304,A -85,B 0,C 180,E1 28061.137,E2 28061.137} C_VEL
LIN {X 0,Y 39.471,Z 994.792,A -85,B 0,C 180,E1 28063.521,E2 28063.521} C_VEL
LIN {X 0,Y 40.252,Z 993.833,A -85,B 0,C 180,E1 28080.048,E2 28080.048} C_VEL
LIN {X 0,Y 43.721,Z 992.931,A -85,B 0,C 180,E1 28096.472,E2 28096.472} C_VEL
LIN {X 0,Y 40.419,Z 993.488,A -85,B 0,C 180,E1 28100.568,E2 28100.568} C_VEL
LIN {X 0,Y 18.261,Z 996.099,A -85,B 0,C 180,E1 28170.007,E2 28170.007} C_VEL
LIN {X 0,Y 35.211,Z 994.227,A -85,B 0,C 180,E1 28234.473,E2 28234.473} C_VEL
LIN {X 0,Y 67.863,Z 987.569,A -85,B 0,C 180,E1 28252.496,E2 28252.496} C_VEL
LIN {X 0,Y 94.817,Z 978.675,A -85,B 0,C 180,E1 28258.247,E2 28258.247} C_VEL
LIN {X 0,Y 60.836,Z 990.02,A -85,B 0,C 180,E1 28265.398,E2 28265.398} C_VEL
LIN {X 0,Y 26.648,Z 996.672,A -85,B 0,C 180,E1 28292.628,E2 28292.628} C_VEL
LIN {X 0,Y 16.634,Z 997.542,A -85,B 0,C 180,E1 28315.877,E2 28315.877} C_VEL
LIN {X 0,Y 14.912,Z 997.057,A -85,B 0,C 180,E1 28407.04,E2 28407.04} C_VEL
LIN {X 0,Y 30.657,Z 995.459,A -85,B 0,C 180,E1 28430.997,E2 28430.997} C_VEL
LIN {X 0,Y 33.596,Z 994.603,A -85,B 0,C 180,E1 28449.52,E2 28449.52} C_VEL
LIN {X 0,Y 31.17,Z 994.832,A -85,B 0,C 180,E1 28453.728,E2 28453.728} C_VEL
LIN {X 0,Y 10.374,Z 996.505,A -85,B 0,C 180,E1 28530.012,E2 28530.012} C_VEL
LIN {X 0,Y 38.363,Z 993.848,A -85,B 0,C 180,E1 28610.661,E2 28610.661} C_VEL
LIN {X 0,Y 60.082,Z 989.742,A -85,B 0,C 180,E1 28617.839,E2 28617.839} C_VEL
LIN {X 0,Y 30.657,Z 995.423,A -85,B 0,C 180,E1 28628.942,E2 28628.942} C_VEL
LIN {X 0,Y 9.836,Z 997.546,A -85,B 0,C 180,E1 28709.987,E2 28709.987} C_VEL
LIN {X 0,Y 14.912,Z 997.057,A -85,B 0,C 180,E1 28767.04,E2 28767.04} C_VEL
LIN {X 0,Y 10.661,Z 997.037,A -85,B 0,C 180,E1 28778.702,E2 28778.702} C_VEL
LIN {X 0,Y 5.733,Z 996.833,A -85,B 0,C 180,E1 28602.25,E2 28602.25} C_VEL
LIN {X 0,Y 8.82,Z 996.659,A -85,B 0,C 180,E1 28608.307,E2 28608.307} C_VEL
LIN {X 0,Y 15.197,Z 996.469,A -85,B 0,C 180,E1 28615.171,E2 28615.171} C_VEL
LIN {X 0,Y 13.613,Z 996.637,A -85,B 0,C 180,E1 28619.857,E2 28619.857} C_VEL
LIN {X 0,Y 1.869,Z 997.136,A -85,B 0,C 180,E1 28709.931,E2 28709.931} C_VEL
LIN {X 0,Y 15.142,Z 996.54,A -85,B 0,C 180,E1 28801.108,E2 28801.108} C_VEL
LIN {X 0,Y 15.19,Z 996.491,A -85,B 0,C 180,E1 28804.712,E2 28804.712} C_VEL
LIN {X 0,Y 2.462,Z 996.913,A -85,B 0,C 180,E1 28890.053,E2 28890.053} C_VEL
LIN {X 0,Y 8.82,Z 996.659,A -85,B 0,C 180,E1 28968.307,E2 28968.307} C_VEL
LIN {X 0,Y 10.812,Z 998.659,A -85,B 0,C 180,E1 28971.344,E2 28971.344} C_VEL
LIN {X 0,Y 10.812,Z 1028,A -85,B 0,C 180,E1 28971.344,E2 28971.344} C_VEL
LIN {X 0,Y 10.812,Z 1028,A -85,B 0,C 180,E1 28971.344,E2 28971.344}

